FUNCTION_BLOCK S_E_C (* Composite Function Block Type *)
  (* Standard: 61499-2 *)
  (* Version 1.0, 2019-04-03, adeel *)
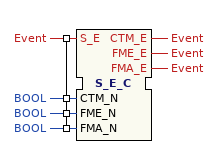
  EVENT_INPUT
    S_E WITH CTM_N, FME_N, FMA_N;
  END_EVENT
  EVENT_OUTPUT
    CTM_E;
    FME_E;
    FMA_E;
  END_EVENT
  VAR_INPUT
    CTM_N : BOOL;
    FME_N : BOOL;
    FMA_N : BOOL;
  END_VAR
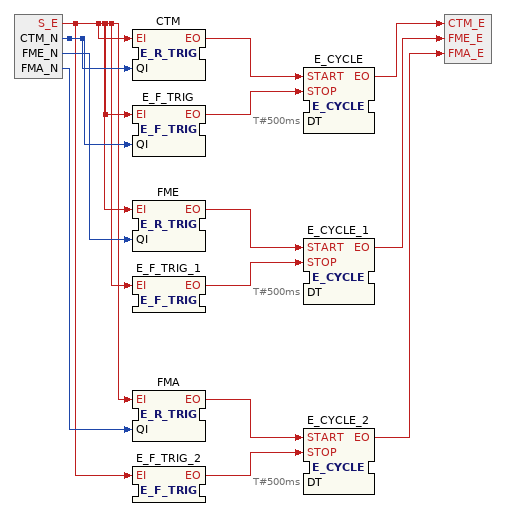
  FBS
    CTM : E_R_TRIG;
    FME : E_R_TRIG;
    FMA : E_R_TRIG;
    E_CYCLE : E_CYCLE(DT := T#500ms);
    E_F_TRIG : E_F_TRIG;
    E_F_TRIG_1 : E_F_TRIG;
    E_F_TRIG_2 : E_F_TRIG;
    E_CYCLE_1 : E_CYCLE(DT := T#500ms);
    E_CYCLE_2 : E_CYCLE(DT := T#500ms);
  END_FBS
  EVENT_CONNECTIONS
    CTM.EO TO E_CYCLE.START;
    E_CYCLE.EO TO CTM_E;
    E_F_TRIG.EO TO E_CYCLE.STOP;
    S_E TO CTM.EI;
    S_E TO E_F_TRIG.EI;
    FME.EO TO E_CYCLE_1.START;
    E_F_TRIG_1.EO TO E_CYCLE_1.STOP;
    FMA.EO TO E_CYCLE_2.START;
    E_F_TRIG_2.EO TO E_CYCLE_2.STOP;
    E_CYCLE_1.EO TO FME_E;
    E_CYCLE_2.EO TO FMA_E;
    S_E TO FME.EI;
    S_E TO E_F_TRIG_1.EI;
    S_E TO FMA.EI;
    S_E TO E_F_TRIG_2.EI;
  END_CONNECTIONS
  DATA_CONNECTIONS
    CTM_N TO CTM.QI;
    FME_N TO FME.QI;
    FMA_N TO FMA.QI;
    CTM_N TO E_F_TRIG.QI;
  END_CONNECTIONS
END_FUNCTION_BLOCK
